PROGRAM SafetyInterface_Enc059
VAR
	{attribute 'TcLinkTo' := '
		.iSafteyCtrlProjectCRC := TIIB[N50S14 (EL6910)]^Device Info Data^Project CRC;
		.iSafetyGroup_State := TIIB[N50S14 (EL6910)]^TwinSAFE Group Info Data^Enc059_SafetyGroup Info Data^State;
		.iSafetyGroup_Diag := TIIB[N50S14 (EL6910)]^TwinSAFE Group Info Data^Enc059_SafetyGroup Info Data^Diag;
		.iSafetyGroup_ComErr := TIIB[N50S14 (EL6910)]^StandardInputs^Enc059_SafetyGroup.oGroup_ComErr_3;
		.iSafetyGroup_ComInStartup := TIIB[N50S14 (EL6910)]^StandardInputs^Enc059_SafetyGroup.oGroup_ComInStartup_4;
		.iSafetyGroup_FBErr := TIIB[N50S14 (EL6910)]^StandardInputs^Enc059_SafetyGroup.oGroup_FBErr_5;
		.iSafetyGroup_FBInRun := TIIB[N50S14 (EL6910)]^StandardInputs^Enc059_SafetyGroup.oGroup_FBInRun_6;
		.iSafetyGroup_InRun := TIIB[N50S14 (EL6910)]^StandardInputs^Enc059_SafetyGroup.oGroup_InRun_7;
		.iSafetyGroup_OtherErr := TIIB[N50S14 (EL6910)]^StandardInputs^Enc059_SafetyGroup.oGroup_OtherErr_8;
		.oSafetyGroup_ErrAck := TIIB[N50S14 (EL6910)]^StandardOutputs^Enc059_SafetyGroup.iGroup_ErrAck_1;
		.oSafetyGroup_Run := TIIB[N50S14 (EL6910)]^StandardOutputs^Enc059_SafetyGroup.iGroup_Run_2;
		.oControlPowerPBLight := TIIB[N50S09 (EL2008)]^Channel 1^Output;
		.iSafetyResetPB := TIIB[N50S14 (EL6910)]^Connection Info Data^Enc059_SafetyGroup.N50S01 Digital 4 In (EL1904)_9 Info Data^Input Safe Data InputChannel3;
		.iEstopPB1_CH1 := TIIB[N50S14 (EL6910)]^Connection Info Data^Enc059_SafetyGroup.N50S01 Digital 4 In (EL1904)_9 Info Data^Input Safe Data InputChannel1;
		.iEstopPB1_CH2 := TIIB[N50S14 (EL6910)]^Connection Info Data^Enc059_SafetyGroup.N50S01 Digital 4 In (EL1904)_9 Info Data^Input Safe Data InputChannel2;
		.iRelayNCContact_Estop := TIIB[N50S14 (EL6910)]^Connection Info Data^Enc059_SafetyGroup.N50S03 Digital 4 In (EL1904)_11 Info Data^Input Safe Data InputChannel1;
		.iSafetyPowerOn_Estop_CH1 := TIIB[N50S14 (EL6910)]^Connection Info Data^Enc059_SafetyGroup.N50S04 Digital 4 Out (EL2904)_20 Info Data^Output Safe Data OutputChannel1;
		.iSafetyPowerOn_Estop_CH2 := TIIB[N50S14 (EL6910)]^Connection Info Data^Enc059_SafetyGroup.N50S04 Digital 4 Out (EL2904)_20 Info Data^Output Safe Data OutputChannel2;
		.iAirPressureOk := TIIB[N50S06 (EL1008)]^Channel 2^Input'}
	fbSafetyInterface : FB_SafetyInterfaceConv;
END_VAR



fbSafetyInterface(
	pSafetyInterface := ADR(gProduced_SafetyInterfaceConv.Enc059));

END_PROGRAM

(* stored: Version 1.1.0.1, ProductVersion 3.1.4024.6
   POU SafetyInterface_Enc059: Id {021ffa31-ebbf-475a-bd47-0103595f8140}, SpecialFunc None *)
